// TIA Portal V16 export
// export: Created 2025-05-30T16:37:07.3427126Z, ExportSetting WithDefaults, DisplayName Totally Integrated Automation Portal, DisplayVersion V16, DisplayName TIA Portal Version Control Interface, DisplayVersion V16, DisplayName TIA Portal Openness, DisplayVersion V16, DisplayName STEP 7 Professional, DisplayVersion V16, DisplayName STEP 7 Safety, DisplayVersion V16, DisplayName WinCC Advanced, DisplayVersion V16
VAR_GLOBAL   // PLC tag table "PositionControl"
   Counter1_IW100 AT %IW100 : Int;
   Counter2_IW102 AT %IW102 : Int;
   "Manual Jog Fwd" AT %M137.0 : Bool;
   "Manual Jog Rev" AT %M137.1 : Bool;
   ReferenceSwitchAxis3 AT %I3.0 : Bool;
   EncoderBand_Alive AT %IW110 : Int;
   EncoderBand_RawCounter AT %IW112 : Int;
   EncoderBand_FineCounter AT %IW113 : Int;
   Zpuls_Encoder_Band AT %I110.3 : Bool;
END_VAR
